PROGRAM MAIN
VAR
END_VAR

popup();

END_PROGRAM

(* stored: Version 1.1.0.1, ProductVersion 3.1.4024.12
   POU MAIN: Id {068e2e2e-5a4f-4ede-b229-3630160c7e8b}, SpecialFunc None *)
